// TIA Portal V17 export
// export: Created 2025-03-05T08:01:21.6954175Z, ExportSetting WithDefaults, DisplayName Totally Integrated Automation Portal, DisplayVersion V17 Update 8, DisplayName TIA Portal Openness, DisplayVersion V17 Update 8, DisplayName TIA Portal Version Control Interface, DisplayVersion V17, DisplayName SINAMICS Startdrive Advanced, DisplayVersion V17 SP2, DisplayName SINAMICS Startdrive G110M, G120, G120C, G120D, G120P, G115D, DisplayVersion V17 SP2, DisplayName SINAMICS Startdrive G130, G150, S120, S150, SINAMICS MV, S210, DisplayVersion V17 SP2, DisplayName STEP 7 Professional, DisplayVersion V17 Update 8, DisplayName SINUMERIK ONE STEP 7 Toolbox, DisplayVersion V17 Update 12, DisplayName SINUMERIK 840D sl STEP 7 Toolbox, DisplayVersion V17 Update 12, DisplayName STEP 7 Safety, DisplayVersion V17 Update 6, DisplayName WinCC Advanced, DisplayVersion V17 Update 8
FUNCTION_BLOCK "FB20201_TRUMPF_GUIDE"   // FB20201, LAD
TITLE = FB20201 GUIDE TRUMPF
{ S7_Optimized_Access := 'FALSE' }
VERSION : 0.1
// stored: AutoNumber false, IsIECCheckEnabled false, SetENOAutomatically false, UDAEnableTagReadback false
   VAR_INPUT
      iEXTERNAL_CONTROL_READY : Bool;
      iLASER_ACTIVE_ON : Bool;
      iMANUAL_START_REQUEST : Bool;
      iAUTO_START_REQUEST : Bool;
      "iMANUAL STOP REQUEST" : Bool;
      "iAUTO STOP REQUEST" : Bool;
      iMACHINE_ON_DELAYED : Bool;
      iSAFETY_GATES_CLOSED_LOCKED : Bool;
      iPILOT_LASER_IS_ON : Bool;
   END_VAR
   VAR_OUTPUT
      oGUIDE_SWITCH_ON : Bool;
      oLASER_POINTER_NOT_READY_ALARM : Bool;
      oSTATION_SEOC_ALARMS : Bool;
      oSwitchoncondition_off : Bool;
      oSwitchoncondition_on : Bool;
      oLimit_right : Bool;
      oLimit_left : Bool;
   END_VAR
   VAR DB_SPECIFIC
      DATA : "LASER POINTER";
      "TIMER FAULT" { S7_SetPoint := 'True'} : TON_TIME;
   END_VAR
   VAR_TEMP
      DB_NUMBER : DInt;
   END_VAR
   VAR CONSTANT
      "FC NUMBER" : Int := 20201;
   END_VAR
   VAR_TEMP   // added for the SCL form of the ladder/FBD networks
      _w1 : Bool;
   END_VAR
BEGIN

NETWORK
TITLE = READ INSTANCE DB NUMBER
      L     DINO;
      +     10#800000;
      T     #DB_NUMBER;

REGION Network 2: START GENERAL CONDITIONS
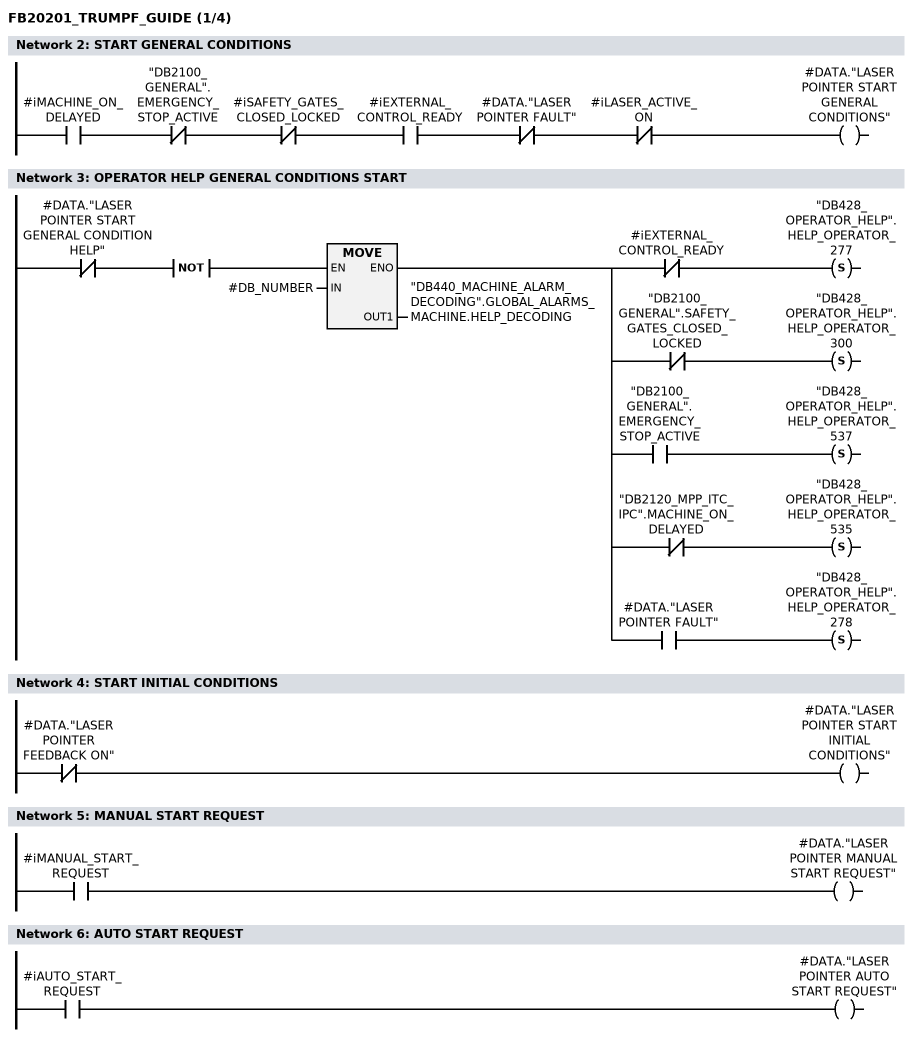
   RUNG wire#powerrail
      Contact( #iMACHINE_ON_DELAYED )
      I_Contact( "DB2100_GENERAL".EMERGENCY_STOP_ACTIVE )
      I_Contact( #iSAFETY_GATES_CLOSED_LOCKED )
      Contact( #iEXTERNAL_CONTROL_READY )
      I_Contact( #DATA."LASER POINTER FAULT" )
      I_Contact( #iLASER_ACTIVE_ON )
      Coil( #DATA."LASER POINTER START GENERAL CONDITIONS" )
   END_RUNG
   // the same network as SCL:
   #DATA."LASER POINTER START GENERAL CONDITIONS" := #iMACHINE_ON_DELAYED AND NOT "DB2100_GENERAL".EMERGENCY_STOP_ACTIVE AND NOT #iSAFETY_GATES_CLOSED_LOCKED AND #iEXTERNAL_CONTROL_READY AND NOT #DATA."LASER POINTER FAULT" AND NOT #iLASER_ACTIVE_ON;
END_REGION

REGION Network 3: OPERATOR HELP GENERAL CONDITIONS START
   RUNG wire#powerrail
      I_Contact( #DATA."LASER POINTER START GENERAL CONDITION HELP" )
      Not()
      Move(in := #DB_NUMBER, out1 => "DB440_MACHINE_ALARM_DECODING".GLOBAL_ALARMS_MACHINE.HELP_DECODING)
      wire#w1
      I_Contact( #iEXTERNAL_CONTROL_READY )
      S_Coil( "DB428_OPERATOR_HELP".HELP_OPERATOR_277 )
   END_RUNG
   RUNG wire#w1
      I_Contact( "DB2100_GENERAL".SAFETY_GATES_CLOSED_LOCKED )
      S_Coil( "DB428_OPERATOR_HELP".HELP_OPERATOR_300 )
   END_RUNG
   RUNG wire#w1
      Contact( "DB2100_GENERAL".EMERGENCY_STOP_ACTIVE )
      S_Coil( "DB428_OPERATOR_HELP".HELP_OPERATOR_537 )
   END_RUNG
   RUNG wire#w1
      I_Contact( "DB2120_MPP_ITC_IPC".MACHINE_ON_DELAYED )
      S_Coil( "DB428_OPERATOR_HELP".HELP_OPERATOR_535 )
   END_RUNG
   RUNG wire#w1
      Contact( #DATA."LASER POINTER FAULT" )
      S_Coil( "DB428_OPERATOR_HELP".HELP_OPERATOR_278 )
   END_RUNG
   // the same network as SCL:
   #_w1 := NOT (NOT #DATA."LASER POINTER START GENERAL CONDITION HELP");
   IF #_w1 THEN "DB440_MACHINE_ALARM_DECODING".GLOBAL_ALARMS_MACHINE.HELP_DECODING := #DB_NUMBER; END_IF;
   IF #_w1 AND NOT #iEXTERNAL_CONTROL_READY THEN "DB428_OPERATOR_HELP".HELP_OPERATOR_277 := TRUE; END_IF;
   IF #_w1 AND NOT "DB2100_GENERAL".SAFETY_GATES_CLOSED_LOCKED THEN
       "DB428_OPERATOR_HELP".HELP_OPERATOR_300 := TRUE;
   END_IF;
   IF #_w1 AND "DB2100_GENERAL".EMERGENCY_STOP_ACTIVE THEN
       "DB428_OPERATOR_HELP".HELP_OPERATOR_537 := TRUE;
   END_IF;
   IF #_w1 AND NOT "DB2120_MPP_ITC_IPC".MACHINE_ON_DELAYED THEN
       "DB428_OPERATOR_HELP".HELP_OPERATOR_535 := TRUE;
   END_IF;
   IF #_w1 AND #DATA."LASER POINTER FAULT" THEN "DB428_OPERATOR_HELP".HELP_OPERATOR_278 := TRUE; END_IF;
END_REGION

REGION Network 4: START INITIAL CONDITIONS
   RUNG wire#powerrail
      I_Contact( #DATA."LASER POINTER FEEDBACK ON" )
      Coil( #DATA."LASER POINTER START INITIAL CONDITIONS" )
   END_RUNG
   // the same network as SCL:
   #DATA."LASER POINTER START INITIAL CONDITIONS" := NOT #DATA."LASER POINTER FEEDBACK ON";
END_REGION

REGION Network 5: MANUAL START REQUEST
   RUNG wire#powerrail
      Contact( #iMANUAL_START_REQUEST )
      Coil( #DATA."LASER POINTER MANUAL START REQUEST" )
   END_RUNG
   // the same network as SCL:
   #DATA."LASER POINTER MANUAL START REQUEST" := #iMANUAL_START_REQUEST;
END_REGION

REGION Network 6: AUTO START REQUEST
   RUNG wire#powerrail
      Contact( #iAUTO_START_REQUEST )
      Coil( #DATA."LASER POINTER AUTO START REQUEST" )
   END_RUNG
   // the same network as SCL:
   #DATA."LASER POINTER AUTO START REQUEST" := #iAUTO_START_REQUEST;
END_REGION

REGION Network 7: GLOBAL START REQUEST
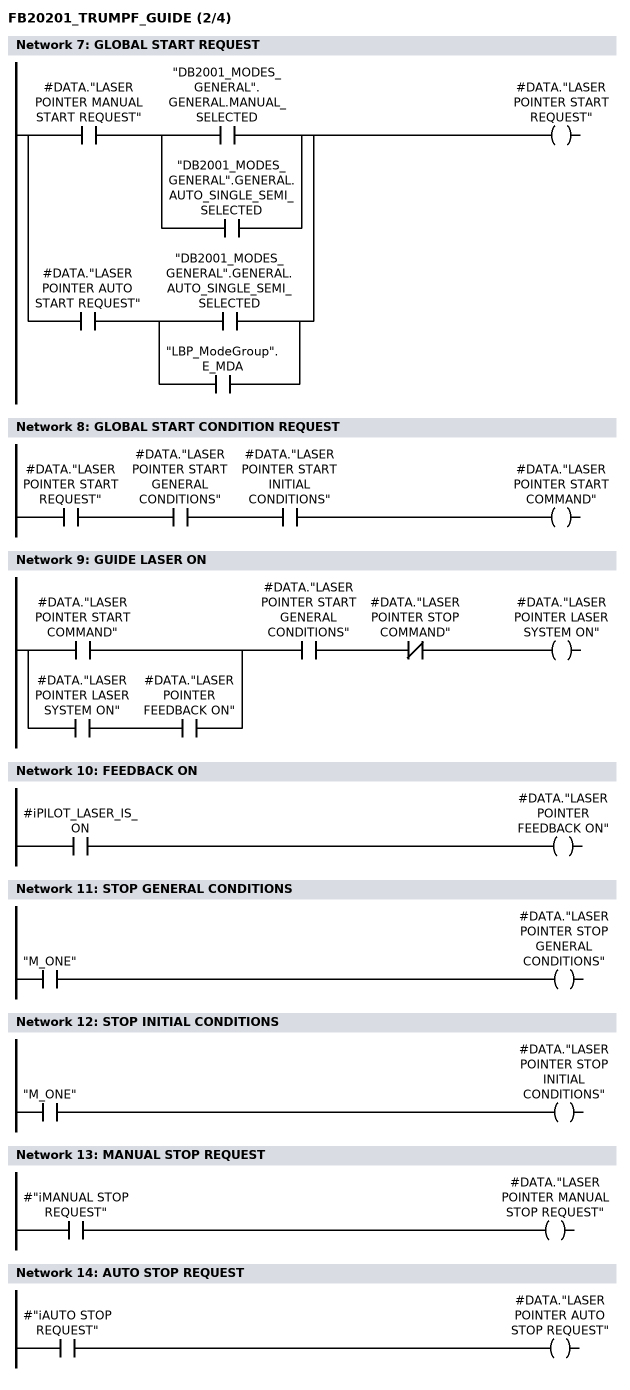
   RUNG wire#powerrail
      Contact( #DATA."LASER POINTER MANUAL START REQUEST" )
      wire#w1
      Contact( "DB2001_MODES_GENERAL".GENERAL.MANUAL_SELECTED )
      wire#w2
      Coil( #DATA."LASER POINTER START REQUEST" )
   END_RUNG
   RUNG wire#w1
      Contact( "DB2001_MODES_GENERAL".GENERAL.AUTO_SINGLE_SEMI_SELECTED )
   END_RUNG wire#w2
   RUNG wire#powerrail
      Contact( #DATA."LASER POINTER AUTO START REQUEST" )
      wire#w3
      Contact( "DB2001_MODES_GENERAL".GENERAL.AUTO_SINGLE_SEMI_SELECTED )
   END_RUNG wire#w2
   RUNG wire#w3
      Contact( "LBP_ModeGroup".E_MDA )
   END_RUNG wire#w2
   // the same network as SCL:
   #DATA."LASER POINTER START REQUEST" := (#DATA."LASER POINTER MANUAL START REQUEST" AND ("DB2001_MODES_GENERAL".GENERAL.MANUAL_SELECTED OR "DB2001_MODES_GENERAL".GENERAL.AUTO_SINGLE_SEMI_SELECTED)) OR (#DATA."LASER POINTER AUTO START REQUEST" AND ("DB2001_MODES_GENERAL".GENERAL.AUTO_SINGLE_SEMI_SELECTED OR "LBP_ModeGroup".E_MDA));
END_REGION

REGION Network 8: GLOBAL START CONDITION REQUEST
   RUNG wire#powerrail
      Contact( #DATA."LASER POINTER START REQUEST" )
      Contact( #DATA."LASER POINTER START GENERAL CONDITIONS" )
      Contact( #DATA."LASER POINTER START INITIAL CONDITIONS" )
      Coil( #DATA."LASER POINTER START COMMAND" )
   END_RUNG
   // the same network as SCL:
   #DATA."LASER POINTER START COMMAND" := #DATA."LASER POINTER START REQUEST" AND #DATA."LASER POINTER START GENERAL CONDITIONS" AND #DATA."LASER POINTER START INITIAL CONDITIONS";
END_REGION

REGION Network 9: GUIDE LASER ON
   RUNG wire#powerrail
      Contact( #DATA."LASER POINTER START COMMAND" )
      wire#w1
      Contact( #DATA."LASER POINTER START GENERAL CONDITIONS" )
      I_Contact( #DATA."LASER POINTER STOP COMMAND" )
      Coil( #DATA."LASER POINTER LASER SYSTEM ON" )
   END_RUNG
   RUNG wire#powerrail
      Contact( #DATA."LASER POINTER LASER SYSTEM ON" )
      Contact( #DATA."LASER POINTER FEEDBACK ON" )
   END_RUNG wire#w1
   // the same network as SCL:
   #DATA."LASER POINTER LASER SYSTEM ON" := (#DATA."LASER POINTER START COMMAND" OR (#DATA."LASER POINTER LASER SYSTEM ON" AND #DATA."LASER POINTER FEEDBACK ON")) AND #DATA."LASER POINTER START GENERAL CONDITIONS" AND NOT #DATA."LASER POINTER STOP COMMAND";
END_REGION

REGION Network 10: FEEDBACK ON
   RUNG wire#powerrail
      Contact( #iPILOT_LASER_IS_ON )
      Coil( #DATA."LASER POINTER FEEDBACK ON" )
   END_RUNG
   // the same network as SCL:
   #DATA."LASER POINTER FEEDBACK ON" := #iPILOT_LASER_IS_ON;
END_REGION

REGION Network 11: STOP GENERAL CONDITIONS
   RUNG wire#powerrail
      Contact( "M_ONE" )
      Coil( #DATA."LASER POINTER STOP GENERAL CONDITIONS" )
   END_RUNG
   // the same network as SCL:
   #DATA."LASER POINTER STOP GENERAL CONDITIONS" := "M_ONE";
END_REGION

REGION Network 12: STOP INITIAL CONDITIONS
   RUNG wire#powerrail
      Contact( "M_ONE" )
      Coil( #DATA."LASER POINTER STOP INITIAL CONDITIONS" )
   END_RUNG
   // the same network as SCL:
   #DATA."LASER POINTER STOP INITIAL CONDITIONS" := "M_ONE";
END_REGION

REGION Network 13: MANUAL STOP REQUEST
   RUNG wire#powerrail
      Contact( #"iMANUAL STOP REQUEST" )
      Coil( #DATA."LASER POINTER MANUAL STOP REQUEST" )
   END_RUNG
   // the same network as SCL:
   #DATA."LASER POINTER MANUAL STOP REQUEST" := #"iMANUAL STOP REQUEST";
END_REGION

REGION Network 14: AUTO STOP REQUEST
   RUNG wire#powerrail
      Contact( #"iAUTO STOP REQUEST" )
      Coil( #DATA."LASER POINTER AUTO STOP REQUEST" )
   END_RUNG
   // the same network as SCL:
   #DATA."LASER POINTER AUTO STOP REQUEST" := #"iAUTO STOP REQUEST";
END_REGION

REGION Network 15: GLOBAL STOP REQUEST
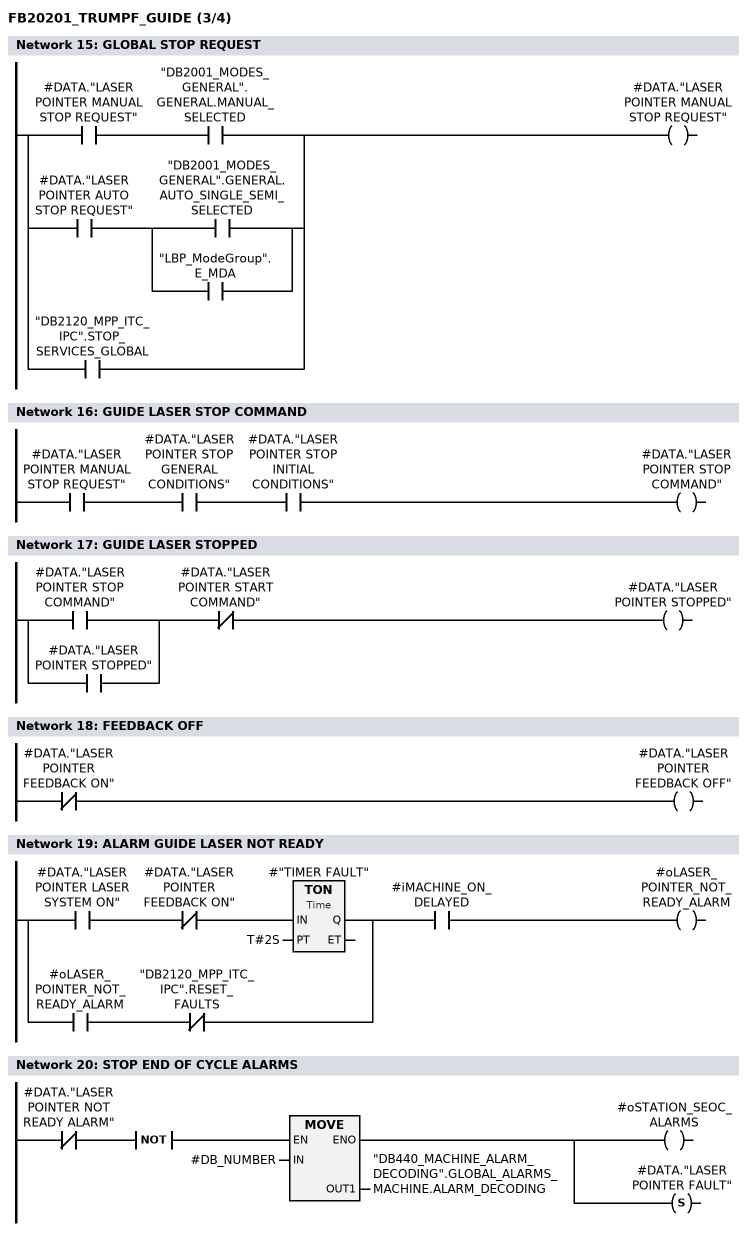
   RUNG wire#powerrail
      Contact( #DATA."LASER POINTER MANUAL STOP REQUEST" )
      Contact( "DB2001_MODES_GENERAL".GENERAL.MANUAL_SELECTED )
      wire#w1
      Coil( #DATA."LASER POINTER MANUAL STOP REQUEST" )
   END_RUNG
   RUNG wire#powerrail
      Contact( #DATA."LASER POINTER AUTO STOP REQUEST" )
      wire#w2
      Contact( "DB2001_MODES_GENERAL".GENERAL.AUTO_SINGLE_SEMI_SELECTED )
   END_RUNG wire#w1
   RUNG wire#w2
      Contact( "LBP_ModeGroup".E_MDA )
   END_RUNG wire#w1
   RUNG wire#powerrail
      Contact( "DB2120_MPP_ITC_IPC".STOP_SERVICES_GLOBAL )
   END_RUNG wire#w1
   // the same network as SCL:
   #DATA."LASER POINTER MANUAL STOP REQUEST" := (#DATA."LASER POINTER MANUAL STOP REQUEST" AND "DB2001_MODES_GENERAL".GENERAL.MANUAL_SELECTED) OR (#DATA."LASER POINTER AUTO STOP REQUEST" AND ("DB2001_MODES_GENERAL".GENERAL.AUTO_SINGLE_SEMI_SELECTED OR "LBP_ModeGroup".E_MDA)) OR "DB2120_MPP_ITC_IPC".STOP_SERVICES_GLOBAL;
END_REGION

REGION Network 16: GUIDE LASER STOP COMMAND
   RUNG wire#powerrail
      Contact( #DATA."LASER POINTER MANUAL STOP REQUEST" )
      Contact( #DATA."LASER POINTER STOP GENERAL CONDITIONS" )
      Contact( #DATA."LASER POINTER STOP INITIAL CONDITIONS" )
      Coil( #DATA."LASER POINTER STOP COMMAND" )
   END_RUNG
   // the same network as SCL:
   #DATA."LASER POINTER STOP COMMAND" := #DATA."LASER POINTER MANUAL STOP REQUEST" AND #DATA."LASER POINTER STOP GENERAL CONDITIONS" AND #DATA."LASER POINTER STOP INITIAL CONDITIONS";
END_REGION

REGION Network 17: GUIDE LASER STOPPED
   RUNG wire#powerrail
      Contact( #DATA."LASER POINTER STOP COMMAND" )
      wire#w1
      I_Contact( #DATA."LASER POINTER START COMMAND" )
      Coil( #DATA."LASER POINTER STOPPED" )
   END_RUNG
   RUNG wire#powerrail
      Contact( #DATA."LASER POINTER STOPPED" )
   END_RUNG wire#w1
   // the same network as SCL:
   #DATA."LASER POINTER STOPPED" := (#DATA."LASER POINTER STOP COMMAND" OR #DATA."LASER POINTER STOPPED") AND NOT #DATA."LASER POINTER START COMMAND";
END_REGION

REGION Network 18: FEEDBACK OFF
   RUNG wire#powerrail
      I_Contact( #DATA."LASER POINTER FEEDBACK ON" )
      Coil( #DATA."LASER POINTER FEEDBACK OFF" )
   END_RUNG
   // the same network as SCL:
   #DATA."LASER POINTER FEEDBACK OFF" := NOT #DATA."LASER POINTER FEEDBACK ON";
END_REGION

REGION Network 19: ALARM GUIDE LASER NOT READY
   RUNG wire#powerrail
      Contact( #DATA."LASER POINTER LASER SYSTEM ON" )
      I_Contact( #DATA."LASER POINTER FEEDBACK ON" )
      { S7_Templates := "time_type := Time" } #"TIMER FAULT".TON(pt := T#2S, et =>)
      wire#w1
      Contact( #iMACHINE_ON_DELAYED )
      Coil( #oLASER_POINTER_NOT_READY_ALARM )
   END_RUNG
   RUNG wire#powerrail
      Contact( #oLASER_POINTER_NOT_READY_ALARM )
      I_Contact( "DB2120_MPP_ITC_IPC".RESET_FAULTS )
   END_RUNG wire#w1
   // the same network as SCL:
   #"TIMER FAULT"(IN := #DATA."LASER POINTER LASER SYSTEM ON" AND NOT #DATA."LASER POINTER FEEDBACK ON",   // TON
                  PT := T#2S);
   #oLASER_POINTER_NOT_READY_ALARM := (#"TIMER FAULT".Q OR (#oLASER_POINTER_NOT_READY_ALARM AND NOT "DB2120_MPP_ITC_IPC".RESET_FAULTS)) AND #iMACHINE_ON_DELAYED;
END_REGION

REGION Network 20: STOP END OF CYCLE ALARMS
   RUNG wire#powerrail
      I_Contact( #DATA."LASER POINTER NOT READY ALARM" )
      Not()
      Move(in := #DB_NUMBER, out1 => "DB440_MACHINE_ALARM_DECODING".GLOBAL_ALARMS_MACHINE.ALARM_DECODING)
      wire#w1
      Coil( #oSTATION_SEOC_ALARMS )
   END_RUNG
   RUNG wire#w1
      S_Coil( #DATA."LASER POINTER FAULT" )
   END_RUNG
   // the same network as SCL:
   #_w1 := NOT (NOT #DATA."LASER POINTER NOT READY ALARM");
   IF #_w1 THEN "DB440_MACHINE_ALARM_DECODING".GLOBAL_ALARMS_MACHINE.ALARM_DECODING := #DB_NUMBER; END_IF;
   #oSTATION_SEOC_ALARMS := #_w1;
   IF #_w1 THEN #DATA."LASER POINTER FAULT" := TRUE; END_IF;
END_REGION

REGION Network 21: LASER SYSTEM FAULT
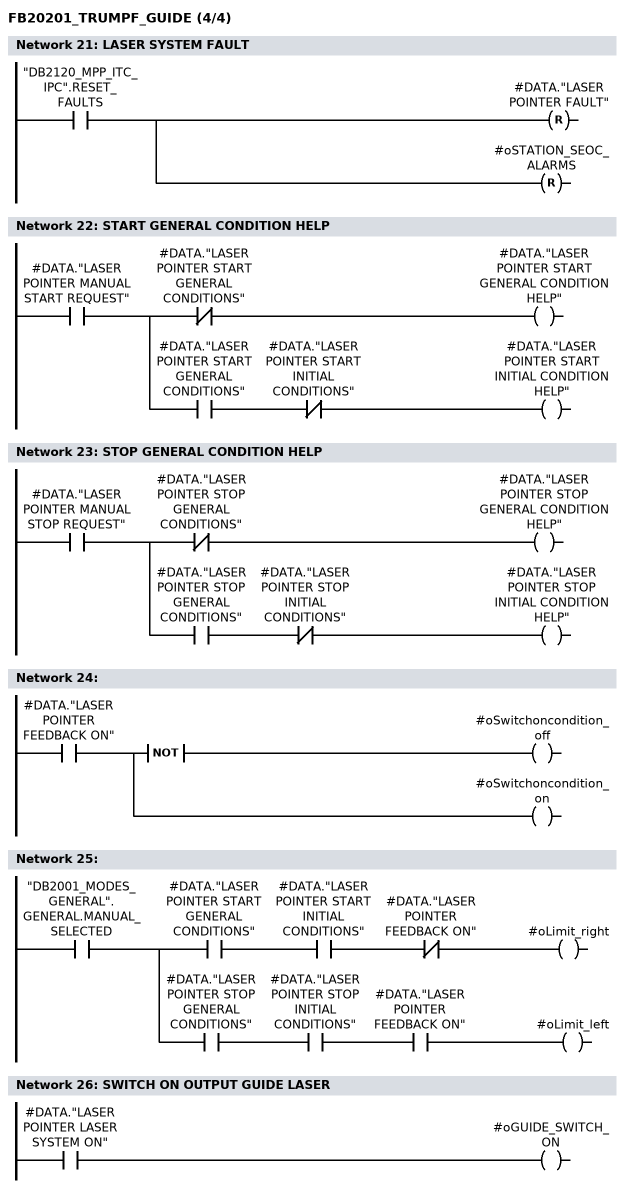
   RUNG wire#powerrail
      Contact( "DB2120_MPP_ITC_IPC".RESET_FAULTS )
      wire#w1
      R_Coil( #DATA."LASER POINTER FAULT" )
   END_RUNG
   RUNG wire#w1
      R_Coil( #oSTATION_SEOC_ALARMS )
   END_RUNG
   // the same network as SCL:
   IF "DB2120_MPP_ITC_IPC".RESET_FAULTS THEN
       #DATA."LASER POINTER FAULT" := FALSE;
       #oSTATION_SEOC_ALARMS := FALSE;
   END_IF;
END_REGION

REGION Network 22: START GENERAL CONDITION HELP
   RUNG wire#powerrail
      Contact( #DATA."LASER POINTER MANUAL START REQUEST" )
      wire#w1
      I_Contact( #DATA."LASER POINTER START GENERAL CONDITIONS" )
      Coil( #DATA."LASER POINTER START GENERAL CONDITION HELP" )
   END_RUNG
   RUNG wire#w1
      Contact( #DATA."LASER POINTER START GENERAL CONDITIONS" )
      I_Contact( #DATA."LASER POINTER START INITIAL CONDITIONS" )
      Coil( #DATA."LASER POINTER START INITIAL CONDITION HELP" )
   END_RUNG
   // the same network as SCL:
   #DATA."LASER POINTER START GENERAL CONDITION HELP" := #DATA."LASER POINTER MANUAL START REQUEST" AND NOT #DATA."LASER POINTER START GENERAL CONDITIONS";
   #DATA."LASER POINTER START INITIAL CONDITION HELP" := #DATA."LASER POINTER MANUAL START REQUEST" AND #DATA."LASER POINTER START GENERAL CONDITIONS" AND NOT #DATA."LASER POINTER START INITIAL CONDITIONS";
END_REGION

REGION Network 23: STOP GENERAL CONDITION HELP
   RUNG wire#powerrail
      Contact( #DATA."LASER POINTER MANUAL STOP REQUEST" )
      wire#w1
      I_Contact( #DATA."LASER POINTER STOP GENERAL CONDITIONS" )
      Coil( #DATA."LASER POINTER STOP GENERAL CONDITION HELP" )
   END_RUNG
   RUNG wire#w1
      Contact( #DATA."LASER POINTER STOP GENERAL CONDITIONS" )
      I_Contact( #DATA."LASER POINTER STOP INITIAL CONDITIONS" )
      Coil( #DATA."LASER POINTER STOP INITIAL CONDITION HELP" )
   END_RUNG
   // the same network as SCL:
   #DATA."LASER POINTER STOP GENERAL CONDITION HELP" := #DATA."LASER POINTER MANUAL STOP REQUEST" AND NOT #DATA."LASER POINTER STOP GENERAL CONDITIONS";
   #DATA."LASER POINTER STOP INITIAL CONDITION HELP" := #DATA."LASER POINTER MANUAL STOP REQUEST" AND #DATA."LASER POINTER STOP GENERAL CONDITIONS" AND NOT #DATA."LASER POINTER STOP INITIAL CONDITIONS";
END_REGION

REGION Network 24
   RUNG wire#powerrail
      Contact( #DATA."LASER POINTER FEEDBACK ON" )
      wire#w1
      Not()
      Coil( #oSwitchoncondition_off )
   END_RUNG
   RUNG wire#w1
      Coil( #oSwitchoncondition_on )
   END_RUNG
   // the same network as SCL:
   #oSwitchoncondition_off := NOT #DATA."LASER POINTER FEEDBACK ON";
   #oSwitchoncondition_on := #DATA."LASER POINTER FEEDBACK ON";
END_REGION

REGION Network 25
   RUNG wire#powerrail
      Contact( "DB2001_MODES_GENERAL".GENERAL.MANUAL_SELECTED )
      wire#w1
      Contact( #DATA."LASER POINTER START GENERAL CONDITIONS" )
      Contact( #DATA."LASER POINTER START INITIAL CONDITIONS" )
      I_Contact( #DATA."LASER POINTER FEEDBACK ON" )
      Coil( #oLimit_right )
   END_RUNG
   RUNG wire#w1
      Contact( #DATA."LASER POINTER STOP GENERAL CONDITIONS" )
      Contact( #DATA."LASER POINTER STOP INITIAL CONDITIONS" )
      Contact( #DATA."LASER POINTER FEEDBACK ON" )
      Coil( #oLimit_left )
   END_RUNG
   // the same network as SCL:
   #oLimit_right := "DB2001_MODES_GENERAL".GENERAL.MANUAL_SELECTED AND #DATA."LASER POINTER START GENERAL CONDITIONS" AND #DATA."LASER POINTER START INITIAL CONDITIONS" AND NOT #DATA."LASER POINTER FEEDBACK ON";
   #oLimit_left := "DB2001_MODES_GENERAL".GENERAL.MANUAL_SELECTED AND #DATA."LASER POINTER STOP GENERAL CONDITIONS" AND #DATA."LASER POINTER STOP INITIAL CONDITIONS" AND #DATA."LASER POINTER FEEDBACK ON";
END_REGION

REGION Network 26: SWITCH ON OUTPUT GUIDE LASER
   RUNG wire#powerrail
      Contact( #DATA."LASER POINTER LASER SYSTEM ON" )
      Coil( #oGUIDE_SWITCH_ON )
   END_RUNG
   // the same network as SCL:
   #oGUIDE_SWITCH_ON := #DATA."LASER POINTER LASER SYSTEM ON";
END_REGION
END_FUNCTION_BLOCK
